# EPICS substitutions: UGARGA.substitutions
file UGARGA.template
{
pattern {S, TA, DN1, DN2}
        {SECAGE, SE, UGA, RGA}
}
